SUBAPPLICATION GreenWhiteBackground3_AXC (* Hintergrundfarbe (TRUE -> Grün, FALSE -> Weiß) für 3 Objekte (AX-Adapter) (Kompakt) *)
  (* Standard: 61499-2 *)
  (* Version 1.0, 2026-07-21, franz, Meisterschulen am Ostbahnhof *)
  PACKAGE MyLib::sys;
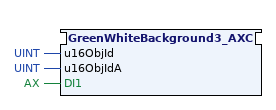
  VAR_INPUT
    u16ObjId : UINT;
    u16ObjIdA : UINT;
  END_VAR
  SOCKETS
    DI1 : adapter::types::unidirectional::AX;
  END_SOCKETS
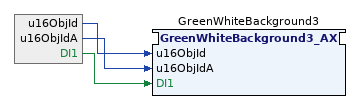
  SUBAPPS
    GreenWhiteBackground3 : MyLib::sys::GreenWhiteBackground3_AX;
  END_SUBAPPS
  DATA_CONNECTIONS
    u16ObjId TO GreenWhiteBackground3.u16ObjId;
    u16ObjIdA TO GreenWhiteBackground3.u16ObjIdA;
  END_CONNECTIONS
  ADAPTER_CONNECTIONS
    DI1 TO GreenWhiteBackground3.DI1;
  END_CONNECTIONS
END_SUBAPPLICATION
